(* CODESYS project RegisterFunctionsInRuntime.project

Project tree, tasks and I/O mapping:
  Device : CoDeSys Control Win V3, 3S - Smart Software Solutions GmbH, version 3.4.2.0
    application Application
      libraries: Standard, 3.4.1.0 (System)
      task MainTask (cyclic, interval t#20ms, priority 1) calls PLC_PRG
      program PLC_PRG [ST]
      function IecFunction1 [ST]
*)

// Device/Application/PLC_PRG
PROGRAM PLC_PRG
VAR
	A : DWORD;
END_VAR

A := IecFunction1(A);

END_PROGRAM

// Device/Application/IecFunction1
{attribute 'register_in_runtime'}
FUNCTION IecFunction1 : DWORD
VAR_INPUT
	dwIn : DWORD;
	
END_VAR
VAR
END_VAR

IecFunction1 := dwIn + 1;

END_FUNCTION
